Fanuc KAREL source: wcntaccel1.kl

PROGRAM wcntaccel1
%NOLOCKGROUP
VAR
  p : POSITION
  q : POSITION
  i : INTEGER
  r : REAL
BEGIN
  WITH $CNT_ACCEL1 = 10 MOVE TO p
END wcntaccel1
